Fanuc KAREL source: DELETE_FILE.kl

PROGRAM T
%NOLOCKGROUP
VAR
 v0 : STRING[40]
 v1 : BOOLEAN
 v2 : INTEGER
BEGIN
 DELETE_FILE(v0, v1, v2)
END T
